Staubli VAL3: SetAccel.pgx

program SetAccel(num value)
begin
  //*******************************************************************************
  //*   ______
  //*  / _____) /|
  //* | |      / /
  //* | | /\  / /
  //* | | \ \/ /  _      Copyright (c) KEOLABS, 2016
  //* | |  \__/  | |        http://www.keolabs.com
  //* | |________| |
  //*  \__________/
  //*
  //********************************************************************************
  //*@file          : SetAccel
  //*@author        : Yves Ragot
  //*@version       : $Id: SetAccel.pgx 1596 2017-01-12 13:28:27Z yves $
  //*@brief         : Change acceleration parameter
  //*
  //*******************************************************************************/

  if ((value > 0) and (value <= 100))
    mNomSpeed.accel = (value * COEFF_ACCEL)
    mNomSpeed.decel = (value * COEFF_ACCEL)
  else
    GeneralStatus = 101
    LastErrorCode = 0
  endIf

end
